(* IEC 61131-3 sources: eCockpitGit/test_project/src, 5 files *)

(* ---- %DUT%alias_test.st ---- *)
TYPE alias_test : INT; END_TYPE

(* ---- %DUT%union_test.st ---- *)
TYPE union_test :
UNION
	union1:BOOL;
	union2:INT;
	union3:WORD;
END_UNION
END_TYPE

(* ---- %GVL%TipsAndTricks.st ---- *)
{attribute 'qualified_only'}
VAR_GLOBAL
END_VAR
(*
//Type Casting is possible
Getting value
value := __CAST(variable,Type);
Setting value
__CAST(variable,Type) := value;
Function Block
__CAST(variable,Function Block Type).value;
Function Block Method
__CAST(variable,Function Block Type).method();

Union variables can have default values by using the var:=(unionMemberName:=value) trick

Thread safe skip, this thread safety makes it so that if two threads access the resource at the same time, the last one will simply skip the action
VAR (Owner)
	block	:DWORD;
END_VAR

IF __COMPARE_AND_SWAP(ADR(block),0,1) THEN
	setValue();
	count			:=		count + 1;
END_IF

Thread safe, this thread safety makes sure that only one thread at a time access a resource, i can intruduce jitter to a calling task if many threads are calling at the same time
VAR (Owner)
	block	:DWORD;
END_VAR

WHILE TRUE DO
	IF __COMPARE_AND_SWAP(ADR(block),0,1) THEN
		doStuff();
		block		:=		0;
		RETURN;
	END_IF
END_WHILE

*)

(* ---- %POU%test.st ---- *)
{"external": false, "compiler_defines": "", "link_always": false, "exclude_from_build": false, "enable_system_call": false}
FUNCTION_BLOCK test
VAR_INPUT
END_VAR
VAR_OUTPUT
END_VAR
VAR
END_VAR

!__IMPLEMENTATION__!

(* ---- %POU%prg_test.st ---- *)
PROGRAM prg_test
VAR
	testVar1:BOOL;
	testVar2:INT;
	testVar3:STRING;

	alias1		:alias_test;
	enum1		:enum_test;
	struct1		:struct_test;
	union1		:union_test;
END_VAR

(*%!%__DELIMITER__%!%*)
IF testVar1 THEN
	testVar2		:=		44;
END_IF

testVar3[4]			:=		testVar2;
